// TIA Portal V18 export
TYPE "UDT_AHUsRegDemand"
// stored: IsFailsafeCompliant false
   STRUCT
      rHeating : Array[1..3] of Real;
      rCooling : Array[1..3] of Real;
      rIAQ : Array[1..3] of Real;
      rBuildingPressure : Array[1..3] of Real;
      rFreshAirTemp : Array[1..3] of Real;
      rFrostProtection : Array[1..3] of Real;
      rFreshAirSummary : Array[1..3] of Real;
   END_STRUCT;
END_TYPE
